(* PLC project Unnamed, Unknown Unnamed 1 *)
(* stored: creationDateTime 2013-01-29T14:01:00, modificationDateTime 2013-02-26T15:59:13 *)

TYPE LOGLEVEL : (CRITICAL, WARNING, INFO, DEBUG) := INFO;
END_TYPE

FUNCTION_BLOCK LOGGER
  VAR_INPUT
    TRIG : BOOL;
    MSG : STRING;
    LEVEL : LOGLEVEL := INFO;
  END_VAR
  VAR
    TRIG0 : BOOL;
  END_VAR

IF TRIG AND NOT TRIG0 THEN
{{
 LogMessage(GetFbVar(LEVEL),(char*)GetFbVar(MSG, .body),GetFbVar(MSG, .len));
}}
END_IF;
TRIG0:=TRIG;

          
END_FUNCTION_BLOCK

FUNCTION_BLOCK DISPLAYMESSAGES
  VAR_INPUT
    TRIG : BOOL;
    MSG1 : STRING;
    MSG2 : STRING;
    MSG3 : STRING;
  END_VAR
  VAR
    TRIG0 : BOOL;
  END_VAR

IF TRIG AND NOT TRIG0 THEN
{{
  setPlcMessages((char*)GetFbVar(MSG1, .body), GetFbVar(MSG1, .len), (char*)GetFbVar(MSG2, .body), GetFbVar(MSG2, .len), (char*)GetFbVar(MSG3, .body), GetFbVar(MSG3, .len));
}}
END_IF;
TRIG0:=TRIG;

          
END_FUNCTION_BLOCK

FUNCTION_BLOCK DISPLAYBUTTONS
  VAR_INPUT
    TRIG : BOOL;
    BTNTEXT1 : STRING;
    BTNCODE1 : INT;
    BTNTEXT2 : STRING;
    BTNCODE2 : INT;
    BTNTEXT3 : STRING;
    BTNCODE3 : INT;
  END_VAR
  VAR
    TRIG0 : BOOL;
  END_VAR

IF TRIG AND NOT TRIG0 THEN
{{
  setPlcButtons((char*)GetFbVar(BTNTEXT1, .body), GetFbVar(BTNTEXT1, .len), GetFbVar(BTNCODE1), (char*)GetFbVar(BTNTEXT2, .body), GetFbVar(BTNTEXT2, .len), GetFbVar(BTNCODE2), (char*)GetFbVar(BTNTEXT3, .body), GetFbVar(BTNTEXT3, .len), GetFbVar(BTNCODE3));
}}
END_IF;
TRIG0:=TRIG;

          
END_FUNCTION_BLOCK

FUNCTION_BLOCK BUTTONPRESSED
  VAR_INPUT
    TRIG : BOOL;
    PROCESSED : BOOL;
  END_VAR
  VAR_OUTPUT
    CODE : INT;
  END_VAR
  VAR
    TRIG0 : BOOL;
  END_VAR

IF TRIG AND NOT TRIG0 THEN
{{
  IF PROCESSED THEN
    CODE:=0;
  END_IF;
  setPlcButtonProcessed(GetFbVar(PROCESSED));
}}
END_IF;
{{
  int32_t code = getPlcButtonPressed();
  SetFbVar(CODE, code);
}}
TRIG0:=TRIG;

          
END_FUNCTION_BLOCK
